FUNCTION_BLOCK RT_E_DELAY (* Delayed propagation of an event-Cancellable *)
  (* Standard: 61499-1; Classification: Event processing *)
  (* Version 0.0, 2008-07-10, 4DIAC-IDE, 4DIAC-Consortium *)
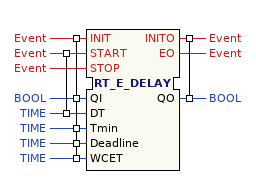
  EVENT_INPUT
    INIT WITH QI, Tmin, Deadline, WCET;
    START WITH DT; (* Begin Delay *)
    STOP; (* Cancel Delay *)
  END_EVENT
  EVENT_OUTPUT
    INITO WITH QO;
    EO; (* Delayed Event *)
  END_EVENT
  VAR_INPUT
    QI : BOOL;
    DT : TIME; (* Delay Time *)
    Tmin : TIME;
    Deadline : TIME;
    WCET : TIME;
  END_VAR
  VAR_OUTPUT
    QO : BOOL;
  END_VAR
END_FUNCTION_BLOCK
